// TwinCAT 3 PLC project examples
// ProgramVersion: 3.1.4026.23
// libraries:
//   rplc, * (TcHaxx)
//   snappy, * (TcHaxx)
//   Tc2_Standard, * (Beckhoff Automation GmbH)
//   Tc2_System, * (Beckhoff Automation GmbH)
//   Tc3_Module, * (Beckhoff Automation GmbH)
//   TcUnit, * (www.tcunit.org)
// project tree:
//   DUTs/ ST_DemoDataType.TcDUT
//   / PlcTaskExamples.TcTTO
//   POUs/ FB_TcUnitExample.TcPOU, FB_TcUnitWithoutSnappyExample.TcPOU, F_CreateDemoData.TcPOU, PRG_TcUnit.TcPOU, PRG_Vanilla.TcPOU

CONFIGURATION examples
    RESOURCE PLC ON TwinCAT3
        TASK PlcTaskExamples(INTERVAL := T#10ms, PRIORITY := 21);
        PROGRAM PRG_Vanilla WITH PlcTaskExamples : PRG_Vanilla;
        PROGRAM PRG_TcUnit WITH PlcTaskExamples : PRG_TcUnit;
    END_RESOURCE
END_CONFIGURATION

// ---- DUTs/ST_DemoDataType.TcDUT
TYPE ST_DemoDataType :
STRUCT
	sString	: STRING;
	nNumber : UDINT;
	fFloat	: REAL;
	aBuffer : ARRAY[0..15] OF BYTE;
END_STRUCT
END_TYPE

// ---- POUs/PRG_Vanilla.TcPOU
PROGRAM PRG_Vanilla
VAR
	fbExample	: FB_Snappy;
		
	eState		: (CONFIG, VERIFY, RESULT) := CONFIG;
	bVerify		: BOOL := FALSE;
	bBuildData  : BOOL := TRUE;
	hr			: HRESULT;
	stDemoDT	: ST_DemoDataType;
	stResult	: ST_VerificationResult;
END_VAR

IF bBuildData THEN
	bBuildData := FALSE;
	stDemoDT := F_CreateDemoData();
END_IF

CASE eState OF
	CONFIG:
		// Configure snappy with defaults:
		// - default JSON serializer (TC3_JsonXml)
		// - default RPC proxy (TcHaxx.rplc)
		// - no test framework, provide testsuite and test name
		hr := fbExample.Configure().UseDefaults().WithoutTestFramework(sTestSuiteName:= 'MyTestSuiteName', sTestName:= 'MyTestName').Build();
		IF SUCCEEDED(hr) THEN
			eState := VERIFY;					
		END_IF
	VERIFY:		
		hr := fbExample.Verify(anyArg:= stDemoDT);
		IF NOT PENDING(hr) THEN
			eState := RESULT;
			bVerify := TRUE;
			stResult := fbExample.stVerificationResult;
		END_IF
	RESULT:
		IF NOT bVerify THEN
			eState := CONFIG;
		END_IF	
END_CASE

END_PROGRAM

// ---- POUs/F_CreateDemoData.TcPOU
FUNCTION F_CreateDemoData : ST_DemoDataType
VAR_INPUT
END_VAR
VAR
	i : UDINT;
END_VAR

F_CreateDemoData.fFloat := -1.23456789;
F_CreateDemoData.nNumber := 16#DEADBEEF;
F_CreateDemoData.sString := 'Lorem ipsum dolor sit amet, consetetur sadipscing elitr, sed diam nonumy';
FOR i:= 0 TO SIZEOF(F_CreateDemoData.aBuffer) DO
	F_CreateDemoData.aBuffer[i] := TO_BYTE(i + 1);
END_FOR

END_FUNCTION

// ---- POUs/PRG_TcUnit.TcPOU
{attribute 'analysis' := '-33'}
PROGRAM PRG_TcUnit
VAR
	fbTcunitExample : FB_TcUnitExample;
	fbNoSnappy		: FB_TcUnitWithoutSnappyExample;
END_VAR



TcUnit.RUN();

END_PROGRAM

// ---- POUs/FB_TcUnitExample.TcPOU
FUNCTION_BLOCK FB_TcUnitExample EXTENDS FB_TestSuite
VAR
	hr				: HRESULT;		
	fbTcUnitAdapter : FB_TcUnitAdapter;
	
	stActual		: ST_DemoDataType;
	{attribute 'analysis' := '-33'}
	stResult		: ST_VerificationResult;
END_VAR

TEST('Test some stuff with TcHaxx.Snappy');

// ARRANGE

// ACT
stActual := F_CreateDemoData();

// ASSERT
hr := fbTcUnitAdapter.Verify(anyArg:= stActual);

IF NOT PENDING(hr) THEN
	TEST_FINISHED_NAMED('Test some stuff with TcHaxx.Snappy');
END_IF

END_FUNCTION_BLOCK

// ---- POUs/FB_TcUnitWithoutSnappyExample.TcPOU
FUNCTION_BLOCK FB_TcUnitWithoutSnappyExample EXTENDS FB_TestSuite
VAR	
	stActual		: ST_DemoDataType;
	stActual2		: ST_DemoDataType;
END_VAR
VAR CONSTANT
	cStringExpected : STRING := 'Lorem ipsum dolor sit amet, consetetur sadipscing elitr, sed diam nonumy';
	cBufferExpected : ARRAY[0..15] OF BYTE := [1,2,3,4,5,6,7,8,9,10,11,12,13,14,15,16];
END_VAR


TEST('Test some stuff without TcHaxx.Snappy');

// ARRANGE

// ACT
stActual := F_CreateDemoData();

// ASSERT
AssertEquals_STRING(Expected:= cStringExpected,
					Actual:= stActual.sString,
					Message:= 'Field sString differs.');
AssertEquals_UDINT(Expected:= 16#DEADBEEF,
					Actual:= stActual.nNumber,
					Message:= 'Field nNumber differs.');
AssertEquals_REAL(Expected:= -1.23456789,
					Actual:= stActual.fFloat,
					Delta:= 0.00001,
					Message:= 'Field fFloat differs.');
AssertArrayEquals_BYTE(Expecteds:= cBufferExpected,
						Actuals:= stActual.aBuffer,
						Message:= 'Field aBuffer differs.');
stActual2 := stActual;						
stActual2.aBuffer[3]:= 55;
AssertEquals(stActual2, stActual, 'Oh snap!');						
TEST_FINISHED_NAMED('Test some stuff without TcHaxx.Snappy');

END_FUNCTION_BLOCK
